FUNCTION_BLOCK FB_Clock
VAR_INPUT
	tPT		: TIME;
END_VAR

VAR_OUTPUT
	bQ		: BOOL;
END_VAR

VAR
	_fbTon1	: TON;
	_fbTon2	: TON;
END_VAR

_fbTon1.PT := tPT;
_fbTon2.PT := tPT;

_fbTon1(IN := NOT bQ);
_fbTon2(IN := bQ);

IF _fbTon1.Q THEN
	bQ := TRUE;
END_IF

IF _fbTon2.Q THEN
	bQ := FALSE;
END_IF

END_FUNCTION_BLOCK

(* stored: Version 1.1.0.1, ProductVersion 3.1.4024.12
   POU FB_Clock: Id {9d8d5595-60d8-0652-1941-c6468040be69}, SpecialFunc None *)
